// TIA Portal project "Training" (V13)

(* hardware
DEVICE "S71500/ET200MP station_1"  S7-1500 station
   slot 0: "Rail_0"  6ES7 590-1***0-0AA0
   slot 1: "PLC_1"  CPU 1516F-3 PN/DP  6ES7 516-3FN00-0AB0  V1.7
   slot 2: "DI 16x24VDC HF_1"  DI 16x24VDC HF  6ES7 521-1BH00-0AB0  V2.0
   slot 3: "AI 8xU/I/RTD/TC ST_1"  AI 8xU/I/RTD/TC ST  6ES7 531-7KF00-0AB0  V2.0
   slot 4: "CP 1543-1_1"  CP 1543-1  6GK7 543-1AX00-0XE0  V1.1
*)

// ===== PLC "PLC_1"  CPU 1516F-3 PN/DP =====

VAR_GLOBAL   // PLC tag table "Default tag table"
   "System_Byte" AT %MB1 : Byte;
   "FirstScan" AT %M1.0 : Bool;
   "DiagStatusUpdate" AT %M1.1 : Bool;
   "AlwaysTRUE" AT %M1.2 : Bool;
   "AlwaysFALSE" AT %M1.3 : Bool;
   "Clock_Byte" AT %MB0 : Byte;
   "Clock_10Hz" AT %M0.0 : Bool;
   "Clock_5Hz" AT %M0.1 : Bool;
   "Clock_2.5Hz" AT %M0.2 : Bool;
   "Clock_2Hz" AT %M0.3 : Bool;
   "Clock_1.25Hz" AT %M0.4 : Bool;
   "Clock_1Hz" AT %M0.5 : Bool;
   "Clock_0.625Hz" AT %M0.6 : Bool;
   "Clock_0.5Hz" AT %M0.7 : Bool;
   "Latch Output" AT %Q50.0 : Bool;
END_VAR

VAR_GLOBAL   // PLC tag table "Local IO Tags"
   "S71500 Green PB" AT %I0.0 : Bool;
   "S71500 Blue PB" AT %I0.1 : Bool;
   "S71500 Pot Upper" AT %IW6 : Int;
   "S71500 Pot Loew" AT %IW14 : Int;
END_VAR

ORGANIZATION_BLOCK "Main"   // OB1, LAD, ProgramCycle
TITLE = "Main Program Sweep (Cycle)"
{ S7_Optimized_Access := 'FALSE' }
VERSION : 0.1
BEGIN

REGION Network 1
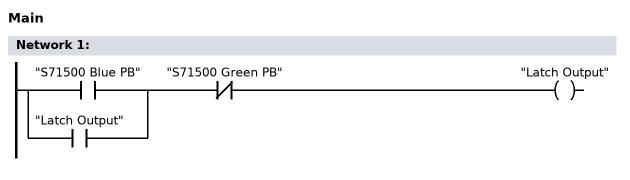
   RUNG wire#powerrail
      Contact( "S71500 Blue PB" )
      wire#w1
      I_Contact( "S71500 Green PB" )
      Coil( "Latch Output" )
   END_RUNG
   RUNG wire#powerrail
      Contact( "Latch Output" )
   END_RUNG wire#w1
   // the same network as SCL:
   "Latch Output" := ("S71500 Blue PB" OR "Latch Output") AND NOT "S71500 Green PB";
END_REGION
END_ORGANIZATION_BLOCK